# EPICS substitutions: kstar/siteApp/TS2/TS2App/Db/ts_result.substitutions
#
file db/TS_RESULT.db
{
    pattern
        { DEV,   ID,    arg,       NAME       }
####################################################
        {"B0",    "0",   "Te",      "CORE1_Te"}
        {"B0",    "1",   "Te",      "CORE2_Te"}
        {"B0",    "2",   "Te",      "CORE3_Te"}

####################################################
        {"B1",    "0",    "Te",      "CORE4_Te"}
        {"B1",    "1",    "Te",      "CORE5_Te"}
        {"B1",    "2",    "Te",      "CORE6_Te"}

#
}
